(* CoDeSys 2.3.9.42 project: _97.pro *)
(* Libraries: C:\Users\bnm\Desktop\oscat_basic_333.lib 25.5.18 09:12:18, Util.lib 18.5.10 15:14:28, Standard.lib 4.10.05 11:14:46, IecSfc.lib 13.4.06 15:51:28, SYSLIBCALLBACK.LIB 26.9.08 15:43:52 *)

(* Global variable list: Global_Variables *)
VAR_GLOBAL
	INPUT: REAL;
	Uroven: REAL;

	reset: BOOL;
	man:BOOL;

	outpid: REAL;

	outpid420: REAL;
	iman: REAL;
	IM1ZADANIE: REAL;
END_VAR

VAR_GLOBAL RETAIN
	shmax: REAL := 17;
	shmin: REAL := 0;
	Ustavka: REAL := 12;
END_VAR

(* POU PLC_PRG, CFC *)
PROGRAM PLC_PRG
VAR
	ln_tr, ln_rt3: LIN_TRAFO;
	PID: CTRL_PID;
	INPUT:REAL;
	KP: REAL;
	TN: REAL;
	TV: REAL;
	ln_rt4: LIN_TRAFO;
	SIGNAL_1: REAL;
	SIGNAL_2: REAL;
	TEMP_ustavka: REAL;
	TEMP_tek: REAL;
END_VAR
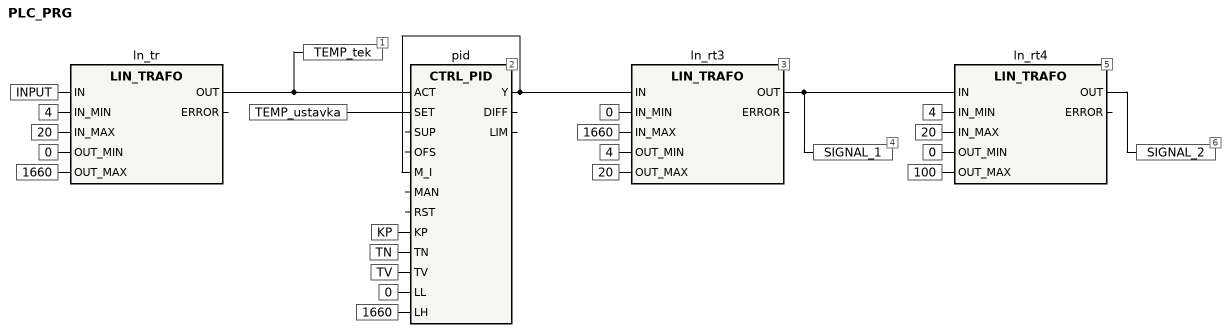
_CFC_ (* Continuous Function Chart, elements in execution order *)
#0 ln_tr:LIN_TRAFO(IN: INPUT, IN_MIN: 4, IN_MAX: 20, OUT_MIN: 0, OUT_MAX: 1660)
#1 TEMP_tek <= #0.OUT
#2 pid:CTRL_PID(ACT: #0.OUT, SET: TEMP_ustavka, SUP: -, OFS: -, M_I: #2.Y, MAN: -, RST: -, KP: KP, TN: TN, TV: TV, LL: 0, LH: 1660)
#3 ln_rt3:LIN_TRAFO(IN: #2.Y, IN_MIN: 0, IN_MAX: 1660, OUT_MIN: 4, OUT_MAX: 20)
#4 SIGNAL_1 <= #3.OUT
#5 ln_rt4:LIN_TRAFO(IN: #3.OUT, IN_MIN: 4, IN_MAX: 20, OUT_MIN: 0, OUT_MAX: 100)
#6 SIGNAL_2 <= #5.OUT
_END_CFC_
(* the same logic as Structured Text *)
ln_tr(IN := INPUT, IN_MIN := 4, IN_MAX := 20, OUT_MIN := 0, OUT_MAX := 1660);
TEMP_tek := ln_tr.OUT;
pid(ACT := ln_tr.OUT, SET := TEMP_ustavka, M_I := pid.Y, KP := KP, TN := TN, TV := TV, LL := 0, LH := 1660);
ln_rt3(IN := pid.Y, IN_MIN := 0, IN_MAX := 1660, OUT_MIN := 4, OUT_MAX := 20);
SIGNAL_1 := ln_rt3.OUT;
ln_rt4(IN := ln_rt3.OUT, IN_MIN := 4, IN_MAX := 20, OUT_MIN := 0, OUT_MAX := 100);
SIGNAL_2 := ln_rt4.OUT;
END_PROGRAM

(* POU PLC_PRG1, CFC *)
PROGRAM PLC_PRG1
VAR
	ctrl1: CTRL_PID;
	KP: REAL;
	TN: REAL;
	TV: REAL;
	ln_tr: LIN_TRAFO;
	ln_tr2: LIN_TRAFO;
	ln_rt3: LIN_TRAFO;
	ln_tr4: LIN_TRAFO;
	ln_tr5: LIN_TRAFO;
	ln_tr6: LIN_TRAFO;
	ln_tr7: LIN_TRAFO;
	ln_tr8: LIN_TRAFO;
	r_tr: R_TRIG;
	f_tr: F_TRIG;
	flag: REAL;
	a:INT;
	ton1: TON;
	ton2: TON;
	test: BOOL;
	r_tr1: R_TRIG;
	sr1: SR;
	tp11: TP;
	CPID: CONTROL_SET2;
	KS: REAL;
	TU: REAL;
	TG: REAL;
	PID_: BOOL;
	KP_: REAL;
	KI: REAL;
	KD: REAL;
	SIN_GEN: GEN;
END_VAR
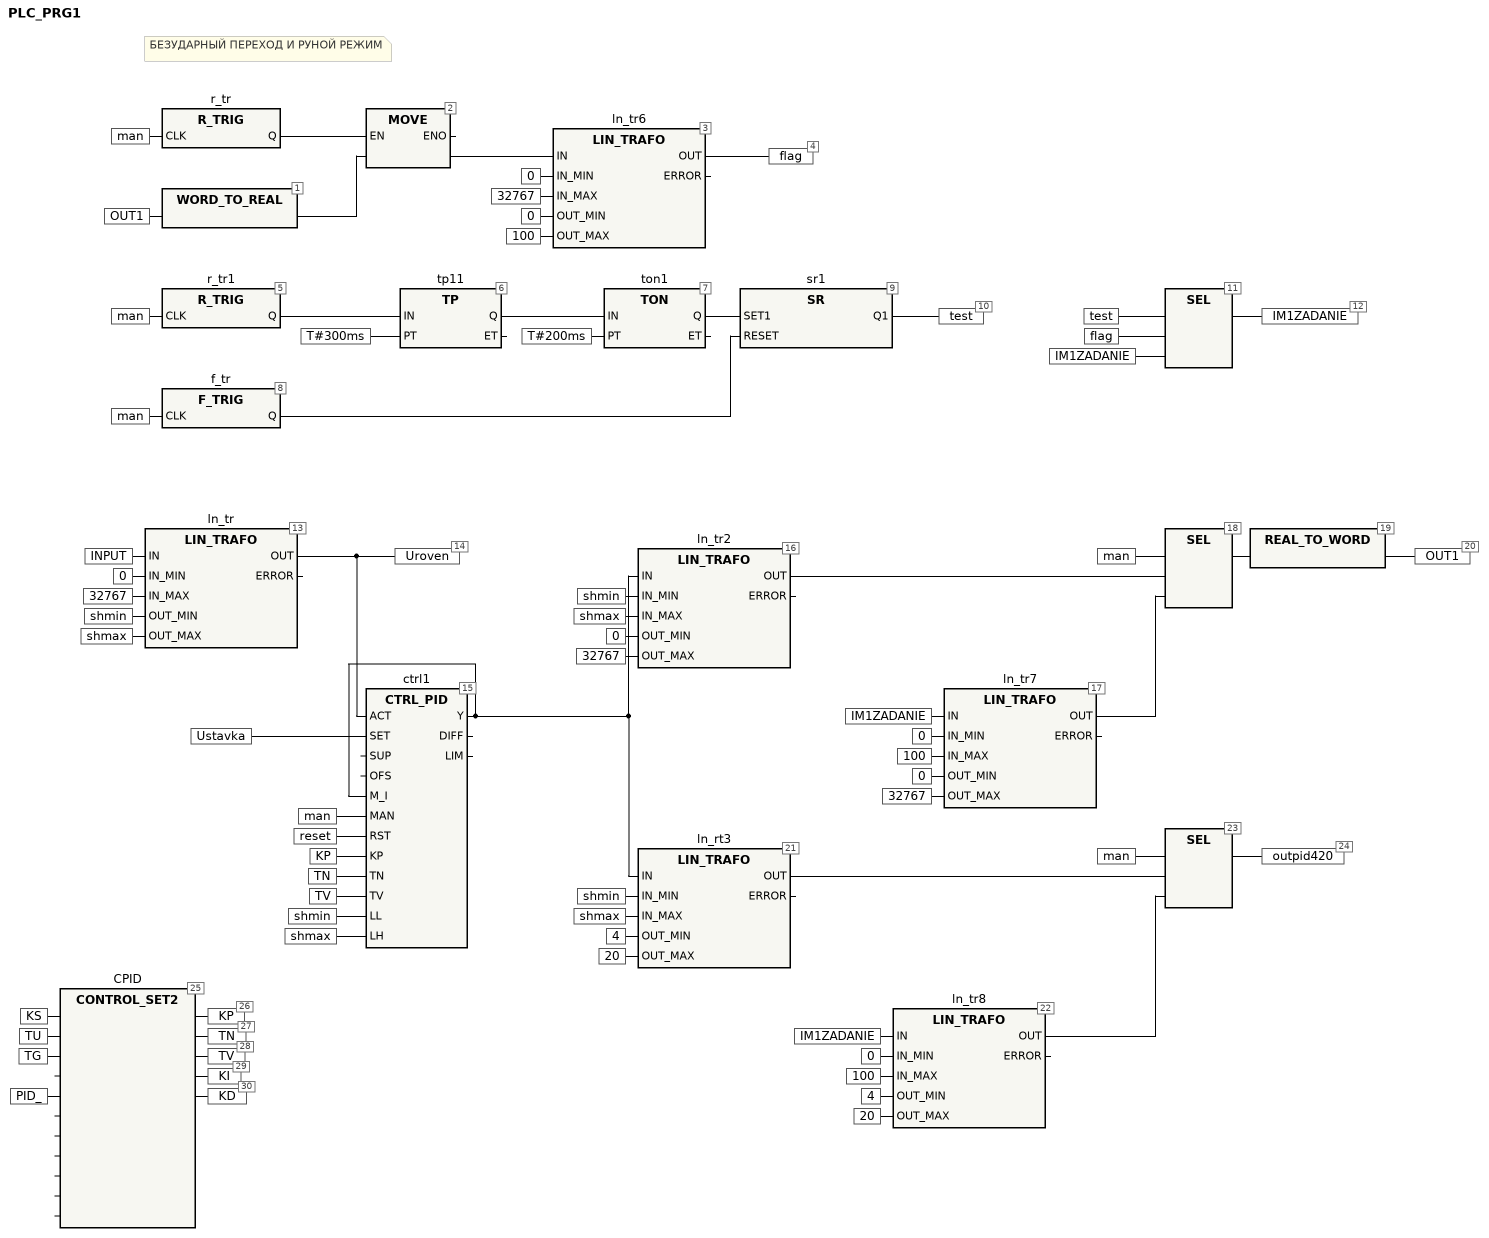
_CFC_ (* Continuous Function Chart, elements in execution order *)
(* БЕЗУДАРНЫЙ ПЕРЕХОД И РУНОЙ РЕЖИМ *)
#0 r_tr:R_TRIG(CLK: man)
#1 WORD_TO_REAL(OUT1)
#2 MOVE(EN: #0.Q, #1)
#3 ln_tr6:LIN_TRAFO(IN: #2, IN_MIN: 0, IN_MAX: 32767, OUT_MIN: 0, OUT_MAX: 100)
#4 flag <= #3.OUT
#5 r_tr1:R_TRIG(CLK: man)
#6 tp11:TP(IN: #5.Q, PT: T#300ms)
#7 ton1:TON(IN: #6.Q, PT: T#200ms)
#8 f_tr:F_TRIG(CLK: man)
#9 sr1:SR(SET1: #7.Q, RESET: #8.Q)
#10 test <= #9.Q1
#11 SEL(test, flag, IM1ZADANIE)
#12 IM1ZADANIE <= #11
#13 ln_tr:LIN_TRAFO(IN: INPUT, IN_MIN: 0, IN_MAX: 32767, OUT_MIN: shmin, OUT_MAX: shmax)
#14 Uroven <= #13.OUT
#15 ctrl1:CTRL_PID(ACT: #13.OUT, SET: Ustavka, SUP: -, OFS: -, M_I: #15.Y, MAN: man, RST: reset, KP: KP, TN: TN, TV: TV, LL: shmin, LH: shmax)
#16 ln_tr2:LIN_TRAFO(IN: #15.Y, IN_MIN: shmin, IN_MAX: shmax, OUT_MIN: 0, OUT_MAX: 32767)
#17 ln_tr7:LIN_TRAFO(IN: IM1ZADANIE, IN_MIN: 0, IN_MAX: 100, OUT_MIN: 0, OUT_MAX: 32767)
#18 SEL(man, #16.OUT, #17.OUT)
#19 REAL_TO_WORD(#18)
#20 OUT1 <= #19
#21 ln_rt3:LIN_TRAFO(IN: #15.Y, IN_MIN: shmin, IN_MAX: shmax, OUT_MIN: 4, OUT_MAX: 20)
#22 ln_tr8:LIN_TRAFO(IN: IM1ZADANIE, IN_MIN: 0, IN_MAX: 100, OUT_MIN: 4, OUT_MAX: 20)
#23 SEL(man, #21.OUT, #22.OUT)
#24 outpid420 <= #23
#25 CPID:CONTROL_SET2(KS, TU, TG, -, PID_, -, -, -, -, -, -)
#26 KP <= #25.out 1
#27 TN <= #25.out 2
#28 TV <= #25.out 3
#29 KI <= #25.out 4
#30 KD <= #25.out 5
_END_CFC_
END_PROGRAM

(* POU PLC_PRG11, CFC *)
PROGRAM PLC_PRG11
VAR
	ctrl1: CTRL_PID;
	KP: REAL;
	TN: REAL;
	TV: REAL;
	ln_tr: LIN_TRAFO;
	ln_tr2: LIN_TRAFO;
	ln_rt3: LIN_TRAFO;
	ln_tr4: LIN_TRAFO;
	ln_tr5: LIN_TRAFO;
	ln_tr6: LIN_TRAFO;
	ln_tr7: LIN_TRAFO;
	ln_tr8: LIN_TRAFO;
	r_tr: R_TRIG;
	f_tr: F_TRIG;
	flag: REAL;
	a:INT;
	ton1: TON;
	ton2: TON;
	test: BOOL;
	r_tr1: R_TRIG;
	sr1: SR;
	tp11: TP;
	CPID: CONTROL_SET2;
	KS: REAL;
	TU: REAL;
	TG: REAL;
	PID_: BOOL;
	KP_: REAL;
	KI: REAL;
	KD: REAL;
	SIN_GEN: GEN;
END_VAR
VAR (* helpers for the ST form of the networks *)
	_t213 : REAL;
END_VAR
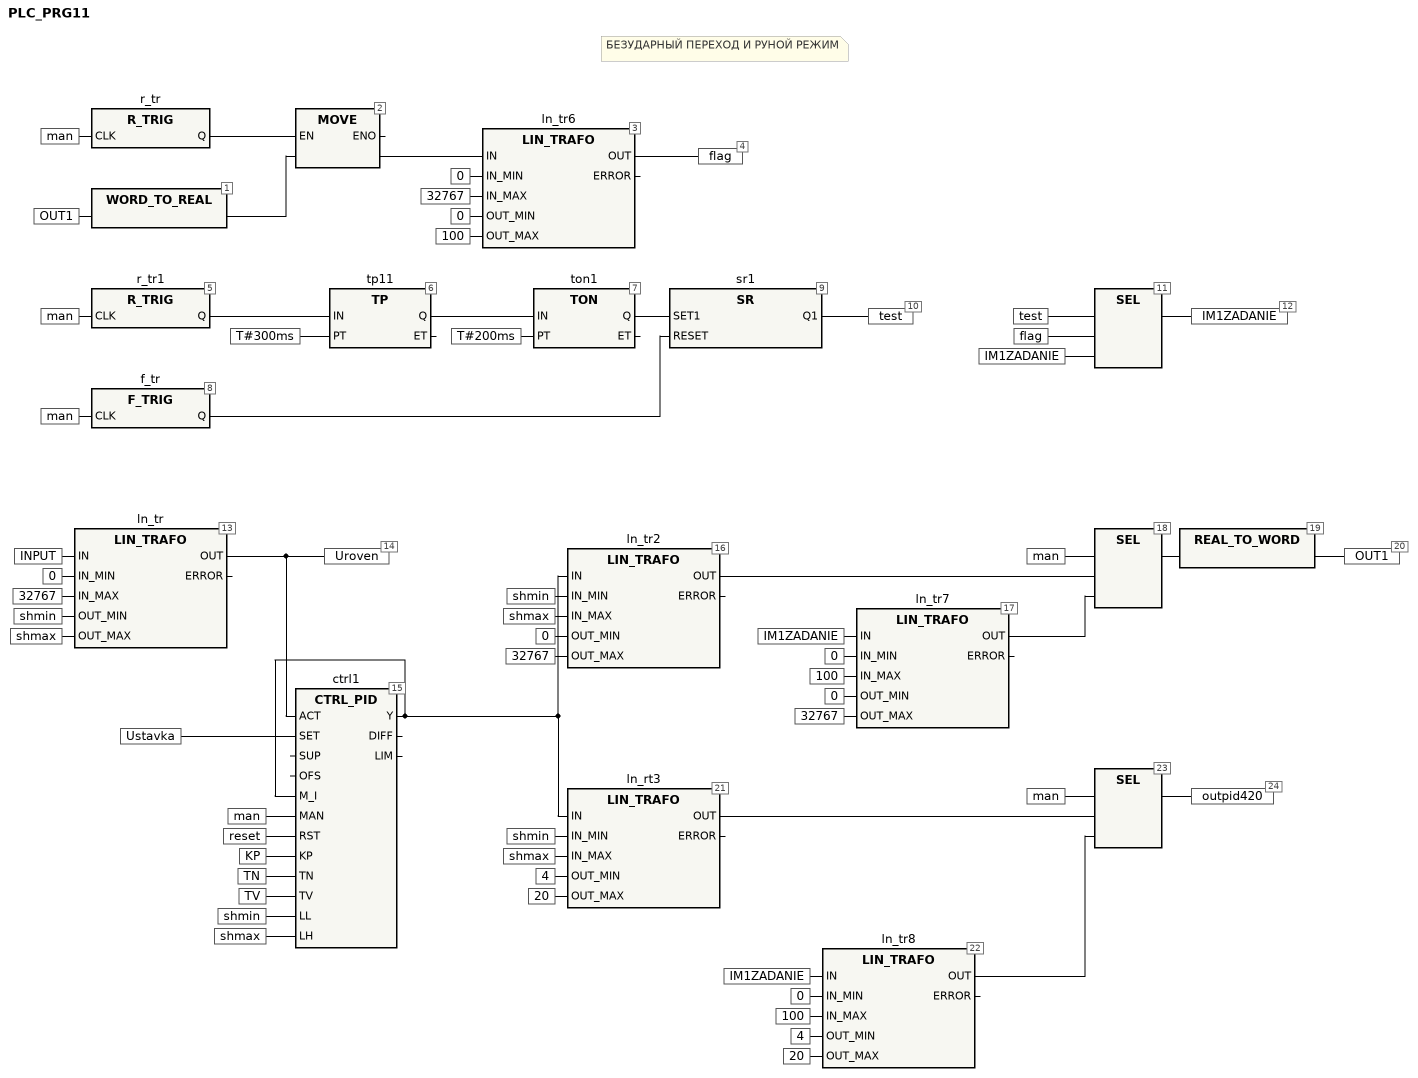
_CFC_ (* Continuous Function Chart, elements in execution order *)
(* БЕЗУДАРНЫЙ ПЕРЕХОД И РУНОЙ РЕЖИМ *)
#0 r_tr:R_TRIG(CLK: man)
#1 WORD_TO_REAL(OUT1)
#2 MOVE(EN: #0.Q, #1)
#3 ln_tr6:LIN_TRAFO(IN: #2, IN_MIN: 0, IN_MAX: 32767, OUT_MIN: 0, OUT_MAX: 100)
#4 flag <= #3.OUT
#5 r_tr1:R_TRIG(CLK: man)
#6 tp11:TP(IN: #5.Q, PT: T#300ms)
#7 ton1:TON(IN: #6.Q, PT: T#200ms)
#8 f_tr:F_TRIG(CLK: man)
#9 sr1:SR(SET1: #7.Q, RESET: #8.Q)
#10 test <= #9.Q1
#11 SEL(test, flag, IM1ZADANIE)
#12 IM1ZADANIE <= #11
#13 ln_tr:LIN_TRAFO(IN: INPUT, IN_MIN: 0, IN_MAX: 32767, OUT_MIN: shmin, OUT_MAX: shmax)
#14 Uroven <= #13.OUT
#15 ctrl1:CTRL_PID(ACT: #13.OUT, SET: Ustavka, SUP: -, OFS: -, M_I: #15.Y, MAN: man, RST: reset, KP: KP, TN: TN, TV: TV, LL: shmin, LH: shmax)
#16 ln_tr2:LIN_TRAFO(IN: #15.Y, IN_MIN: shmin, IN_MAX: shmax, OUT_MIN: 0, OUT_MAX: 32767)
#17 ln_tr7:LIN_TRAFO(IN: IM1ZADANIE, IN_MIN: 0, IN_MAX: 100, OUT_MIN: 0, OUT_MAX: 32767)
#18 SEL(man, #16.OUT, #17.OUT)
#19 REAL_TO_WORD(#18)
#20 OUT1 <= #19
#21 ln_rt3:LIN_TRAFO(IN: #15.Y, IN_MIN: shmin, IN_MAX: shmax, OUT_MIN: 4, OUT_MAX: 20)
#22 ln_tr8:LIN_TRAFO(IN: IM1ZADANIE, IN_MIN: 0, IN_MAX: 100, OUT_MIN: 4, OUT_MAX: 20)
#23 SEL(man, #21.OUT, #22.OUT)
#24 outpid420 <= #23
_END_CFC_
(* the same logic as Structured Text *)
(* БЕЗУДАРНЫЙ ПЕРЕХОД И РУНОЙ РЕЖИМ *)
r_tr(CLK := man);
IF r_tr.Q THEN _t213 := WORD_TO_REAL(OUT1); END_IF;
ln_tr6(IN := _t213, IN_MIN := 0, IN_MAX := 32767, OUT_MIN := 0, OUT_MAX := 100);
flag := ln_tr6.OUT;
r_tr1(CLK := man);
tp11(IN := r_tr1.Q, PT := T#300ms);
ton1(IN := tp11.Q, PT := T#200ms);
f_tr(CLK := man);
sr1(SET1 := ton1.Q, RESET := f_tr.Q);
test := sr1.Q1;
IM1ZADANIE := SEL(test, flag, IM1ZADANIE);
ln_tr(IN := INPUT, IN_MIN := 0, IN_MAX := 32767, OUT_MIN := shmin, OUT_MAX := shmax);
Uroven := ln_tr.OUT;
ctrl1(ACT := ln_tr.OUT, SET := Ustavka, M_I := ctrl1.Y, MAN := man, RST := reset, KP := KP, TN := TN, TV := TV, LL := shmin, LH := shmax);
ln_tr2(IN := ctrl1.Y, IN_MIN := shmin, IN_MAX := shmax, OUT_MIN := 0, OUT_MAX := 32767);
ln_tr7(IN := IM1ZADANIE, IN_MIN := 0, IN_MAX := 100, OUT_MIN := 0, OUT_MAX := 32767);
OUT1 := REAL_TO_WORD(SEL(man, ln_tr2.OUT, ln_tr7.OUT));
ln_rt3(IN := ctrl1.Y, IN_MIN := shmin, IN_MAX := shmax, OUT_MIN := 4, OUT_MAX := 20);
ln_tr8(IN := IM1ZADANIE, IN_MIN := 0, IN_MAX := 100, OUT_MIN := 4, OUT_MAX := 20);
outpid420 := SEL(man, ln_rt3.OUT, ln_tr8.OUT);
END_PROGRAM

(* Visualisation mn
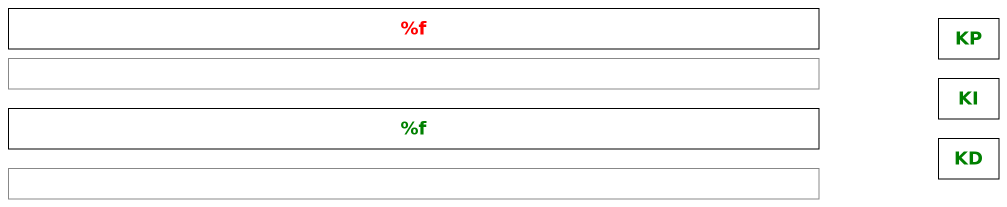
rectangle at (90,30)-(901,71): text "%f"; shows PLC_PRG.TEMP_tek
rectangle at (90,130)-(901,171): text "%f"; shows PLC_PRG.TEMP_ustavka
rounded rectangle at (1020,40)-(1081,81): text "KP"
rounded rectangle at (1020,100)-(1081,141): text "KI"
rounded rectangle at (1020,160)-(1081,201): text "KD"
2 more shapes without text or variables
5 elements of other kinds (tables, trends, ...) not read
*)
